// TIA Portal V20 export
// export: Created 2026-07-10T11:12:25.9327932Z, ExportSetting WithDefaults, DisplayName Totally Integrated Automation Portal, DisplayVersion V20, DisplayName TIA Portal Openness, DisplayVersion V20, DisplayName TIA Portal Version Control Interface, DisplayVersion V20, DisplayName STEP 7 Professional, DisplayVersion V20, DisplayName STEP 7 Safety, DisplayVersion V20, DisplayName WinCC Basic/Comfort/Advanced, DisplayVersion V20, DisplayName WinCC Unified, DisplayVersion V20
FUNCTION_BLOCK "MBServer"   // FB19, SCL
{ S7_Optimized_Access := 'TRUE' }
VERSION : 0.1
// stored: AutoNumber true, IsIECCheckEnabled false, IsRetainMemResEnabled false, MemoryReserve 100, SetENOAutomatically false, UDAEnableTagReadback false
BEGIN
   "MB_SERVER_DB"(DISCONNECT:=FALSE,
                  NDR=>"MB_Config".NDR,
                  DR=>"MB_Config".DR,
                  ERROR=>"MB_Config".ERROR,
                  MB_HOLD_REG:="MB".Table,
                  CONNECT:="MB_Config".CONNECT);
END_FUNCTION_BLOCK
